(* IEC 61131-3 sources: SRCI/RobotLibrary/RobotLibrary/Interfaces, 2 files *)

(* ---- IMessageLogger.st ---- *)
INTERFACE IMessageLogger

METHOD AddMessageLog
VAR_INPUT
  /// Message to add to the log
  MessageLog : AlarmMessage;
END_VAR

END_METHOD

METHOD AddSystemLog
VAR_INPUT
  /// System messafe to add to the log
  SystemLog : STRING(255);
END_VAR

END_METHOD

(* ---- IRobotLibraryCommandFB.st ---- *)
INTERFACE IRobotLibraryCommandFB

METHOD PUBLIC CallBack : DINT
VAR_INPUT
  /// Response data
  RspData : AxesGroupAcyclicAcrEntryRspBuffer;
END_VAR

END_METHOD

PROPERTY CommandData : SendData

GET

END_GET

SET

END_SET
